PROGRAM testProg
VAR

END_VAR

//Initial parameters of an Axis
IF _TaskInfo[fbGetCurTaskIndex.index].FirstCycle THEN
    //Initial default values:
    GVL.astAxes[1].stInputs.bLimitBwd := 1;
    GVL.astAxes[1].stInputs.bLimitFwd := 1;
    GVL.astAxes[1].stControl.bEnable := 1;
    GVL.astAxes[2].stInputs.bLimitBwd := 1;
    GVL.astAxes[2].stInputs.bLimitFwd := 1;
    GVL.astAxes[2].stControl.bEnable := 1;
END_IF

END_PROGRAM

(* stored: Version 1.1.0.1, ProductVersion 3.1.4024.0
   POU testProg: Id {1a43acb4-bd2e-4637-97fb-9976d47292b6}, SpecialFunc None *)
